INTERFACE I_SysLogListener

METHOD OnTraceReceived
VAR_INPUT
    Message : ST_SysLogMessages;
END_VAR
END_METHOD

END_INTERFACE

(* stored: Version 1.1.0.1
   Itf I_SysLogListener: Id {b46ba456-5ae1-4c47-8197-f2528ac4dd97}
   Method OnTraceReceived: Id {ecb04e39-5a33-41e2-ab97-d56f2aed52c4} *)
